(* CODESYS project EX2.project

Project tree, tasks and I/O mapping:
  Device : CODESYS Control Win V3, 3S - Smart Software Solutions GmbH, order no. 305021, version 3.5.11.30
    application Application
      libraries: Standard, * (System)
      task MainTask (cyclic, interval t#20ms, priority 1) calls PLC_PRG
      task VISU_TASK (cyclic, interval 100 ms, priority 31) calls VisuElems.Visu_Prg
      program PLC_PRG [LD]
      visualisation Visualization
  libraries: VisuSymbols, 3.5.10.0 (System)
  text list GlobalTextList
*)

// Device/Application/PLC_PRG
PROGRAM PLC_PRG
VAR
	BT1 : BOOL;          // LIGA L1
	BT2 : BOOL;          // LIGA L2
	BT3 : BOOL;          // LIGA L3
	L1 : BOOL;           // LAMPADA L1
	L2 : BOOL;           // LAMPADA L2
	L3 : BOOL;           // LAMPADA L3
END_VAR
VAR // added by the converter: edge detectors and wires of the graphical bodies
    _rt1, _rt2, _rt3 : R_TRIG;
    _ft1, _ft2, _ft3 : F_TRIG;
END_VAR

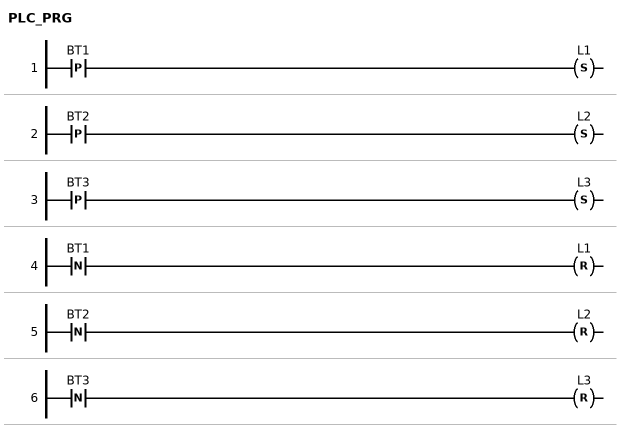
// NETWORK 1
_rt1(CLK := BT1);
L1 S= _rt1.Q;

// NETWORK 2
_rt2(CLK := BT2);
L2 S= _rt2.Q;

// NETWORK 3
_rt3(CLK := BT3);
L3 S= _rt3.Q;

// NETWORK 4
_ft1(CLK := BT1);
L1 R= _ft1.Q;

// NETWORK 5
_ft2(CLK := BT2);
L2 R= _ft2.Q;

// NETWORK 6
_ft3(CLK := BT3);
L3 R= _ft3.Q;

END_PROGRAM

// Device/Application/Visualization
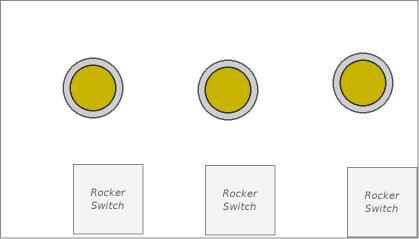
VISUALIZATION Visualization  // 419x239
    Lamp1 (58,53 70x70), variable: PLC_PRG.L1, style: Lamp-Lamp1-Yellow
    Lamp1 (193,55 70x70), variable: PLC_PRG.L2, style: Lamp-Lamp1-Yellow
    Lamp1 (328,48 70x70), variable: PLC_PRG.L3, style: Lamp-Lamp1-Yellow
    RockerSwitch (73,164 70x70), variable: PLC_PRG.BT1, behaviour: TOGGLE, style: Switch-RockerSwitch-Gray
    RockerSwitch (205,165 70x70), variable: PLC_PRG.BT2, behaviour: TOGGLE, style: Switch-RockerSwitch-Gray
    RockerSwitch (347,167 70x70), variable: PLC_PRG.BT3, behaviour: TOGGLE, style: Switch-RockerSwitch-Gray
END_VISUALIZATION
